TYPE SensorConfiguration EXTENDS BaseConfiguration:
STRUCT
	sReturnType : STRING;
	sType : STRING;
	sSensPosition : STRING;
	iSensIndex : DINT;
END_STRUCT
END_TYPE

(* stored: Version 1.1.0.1
   DUT SensorConfiguration: Id {84110889-d2dc-4143-a45b-c9c45971aad3} *)
